// TwinCAT 3 PLC project Example
// ProgramVersion: 3.1.4024.12
// libraries:
//   Struckig, * (Struckig)
//   Tc2_Standard, * (Beckhoff Automation GmbH)
//   Tc2_System, * (Beckhoff Automation GmbH)
//   Tc3_Module, * (Beckhoff Automation GmbH)
// project tree:
//   / PlcTask.TcTTO
//   POUs/ MAIN.TcPOU
// real-time tasks:
//   TASK PlcTask: cycle T#1ms, priority 20, ADS port 350

CONFIGURATION Example
    RESOURCE PLC ON TwinCAT3
        TASK PlcTask(INTERVAL := T#1ms, PRIORITY := 20);
        PROGRAM MAIN WITH PlcTask : MAIN;
    END_RESOURCE
END_CONFIGURATION

// ---- POUs/MAIN.TcPOU
PROGRAM MAIN
VAR
  ruckig : Ruckig(0.001);
  input : InputParameterStruct;
  output : OutputParameterStruct;    
  init : BOOL := TRUE;
END_VAR

IF init
THEN
  init := FALSE;

  input.dofs := 1;
  input.enabled[0] := TRUE;
  input.max_velocity[0] := 1.2;
  input.max_acceleration[0] := 4.0;
  input.max_jerk[0] := 10;
  
  input.current_position[0] := 0;
  input.current_velocity[0] := 0;
  input.current_acceleration[0] := 0;
  
  input.target_position[0] := 1;
  input.target_velocity[0] := 0;
  input.target_acceleration[0] := 0;  
END_IF

ruckig.update(input, output);
input.current_position := output.new_position;
input.current_velocity := output.new_velocity;
input.current_acceleration := output.new_acceleration;

END_PROGRAM
